RoboDK station: Project.rdk

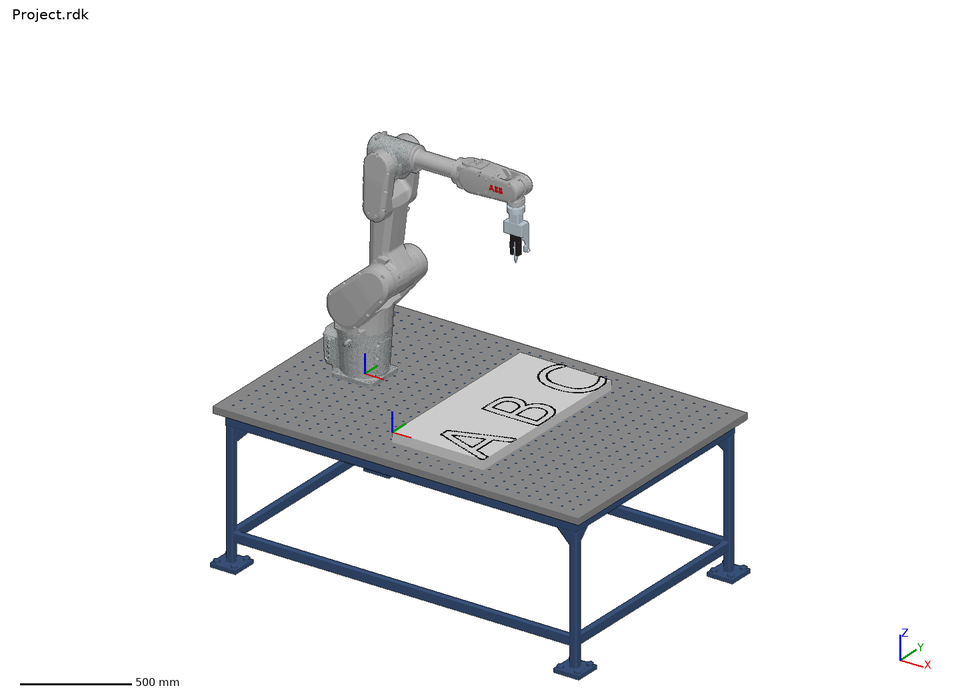
[picture v0: the station drawn from its stored meshes, robots at their saved joint values, targets as dots, program paths as lines]
Station Project (saved by RoboDK 5.5.2). Poses are relative to the parent item; angles as X-Y-Z fixed-axis rotations.
  - object Table at (0, 0, 0) mm, size 2020 x 1340 x 800 mm, geometry from Table-2000x1200x800mm.sld
  - frame Robot_Base at (0, 0, 0) mm
    - robot Robot (model ABB IRB 1300-7/1.4): 6 axes, payload 7 kg, reach 1400 mm, repeatability 0.02 mm, weight 78.5 kg
        modified DH rows (alpha deg, a mm, theta deg, d mm): 0, 0, 0, 544; -90, 150, -90, 0; 0, 575, 0, 0; -90, 40, 0, 675; 90, 0, 0, 0; -90, 0, 180, 90
        joint limits [-180, -95, -210, -230, -130, -400] to [180, 155, 69, 230, 130, 400]; home [0, 0, 0, 0, 0, 0]; saved at [0, 0, 0, 0, 90, 0]
      - tool Pencil, TCP at (0, 0, 283) mm, size 100 x 89.2 x 281.5 mm
    - object pixel at (0, 0, 0) mm, size 10 x 10 x 1 mm
    - frame Board_Frame at (500, -500, 50) mm
      - object Paper_Pixel at (0, 0, 0) mm, size 250 x 250 x 50 mm
      - object Papers at (0, 0, 0) mm, size 505.1 x 1012 x 51 mm
  - Python program main (listed below)

--- Python program main ---
#!/usr/bin/python

# Type help("robodk.robolink") or help("robodk.robomath") for more information
# Press F5 to run the script
# Documentation: https://robodk.com/doc/en/RoboDK-API.html
# Reference:     https://robodk.com/doc/en/PythonAPI/robodk.html
# Note: It is not required to keep a copy of this file, your Python script is saved with your RDK project

# RoboWriter class is a sample class for writing robot.
# For now it assumes that the writing board lies within the robot dextrous workspace

# Import the APIs (RoboDK and Robolink)
from robodk import *
from robolink import *

import sys
import os
import re

SIZE_BOARD = [500, 1000]     # Size of the image. The image will be scaled keeping its aspect ratio
MM_X_PIXEL = 10             # in mm. The path will be cut depending on the pixel size. If this value is changed it is recommended to scale the pixel object

TEXT_SVG='images/test.svg'

class RoboWriter:
    def __init__(self):
        RDK = Robolink()    # Open connection with Robolink library

        # get the robot, frame and tool objects
        self.robot = RDK.Item('', ITEM_TYPE_ROBOT)  # Get the first robot
        self.Board_Frame = RDK.Item('Board_Frame')  # Get the Board_frame
        self.Pencil = RDK.Item('Pencil')            # Get the Pencil

        self.pixel = RDK.Item('pixel')  # get the pixel reference to draw

        image = RDK.Item('Papers')                                   # Get the Paper
        if image.Valid() and image.Type() == ITEM_TYPE_OBJECT:          # If something is already written on the board erase it.
            image.Delete()

        board_pixel = RDK.Item('Paper_Pixel')   # Get the White Board (The display board will be traced using this board)
        # Create Display Board. Difference between White Board and Display board is that
        # White board is a small sized pixel that will be replicated on Display board to
        # show the image

        # Create Display board
        board_pixel.Copy()  # Create a copy of blackboard
        self.board = self.Board_Frame.Paste()   # Create a board with Board Frame as reference frame
        self.board.setVisible(True, False)  # Set the visibility of the board
        self.board.setName('Papers') # Name the board as Display Board

    def write(self, content):
        APPROACH = 100  # approach distance in MM for each path

        home_joints = self.robot.JointsHome().tolist() #[0,0,0,0,90,0] # home joints, in deg
        if abs(home_joints[4]) < 5:
            home_joints[4] = 90.0
        #home_joints[5] = 180

        self.robot.setPoseFrame(self.Board_Frame)
        self.robot.setPoseTool(self.Pencil)
        self.robot.MoveJ(home_joints)   # Move robot to home configuration

        # Get the target orientation depending on the tool orientation at home position
        board_frame_pose = self.Board_Frame.Pose() # Board Frame Pose wrt Robot Base
        robot_flange_pose = self.robot.SolveFK(home_joints) # Robot Flange Pose wrt Robot Base
        TCP_pose = self.Pencil.Pose()   # TCP Pose wrt Flange
        # Use trandformation to get the target orientation wrt Tool
        T2T_Orientation = invH(board_frame_pose)*robot_flange_pose*TCP_pose
        T2T_Orientation[0:3,3] = Mat([0,0,0]) # Set translation to 0

        size_img = content.size_poly()  # returns the size of the current polygon
        self.board.Scale([SIZE_BOARD[0]/250, SIZE_BOARD[1]/250, 1]) # adjust the board size to the image size (scale)

        for path in content:
            # use the pixel reference to set the path color, set pixel width and copy as a reference
            self.pixel.Recolor(path.fill_color)
            data_points_in_current_path = path.nPoints()

            # robot movement: approach to the first target
            initial_target = path.getPoint(0)
            target0 = transl(SIZE_BOARD[0]-initial_target.x, initial_target.y, 0)*T2T_Orientation
            target0_app = target0*transl(0,0,-APPROACH)
            self.robot.MoveL(target0_app)

            for i in range(data_points_in_current_path):
                p_i = path.getPoint(i)
                v_i = path.getVector(i)
                pt_pose = transl(SIZE_BOARD[0]-p_i.x, p_i.y, 0)*rotz(v_i.angle())

                target = transl(SIZE_BOARD[0]-p_i.x, p_i.y, 0)*(T2T_Orientation)

                # Move the robot to the next target
                self.robot.MoveL(target)

                # create a new pixel object with the calculated pixel pose
                self.board.AddGeometry(self.pixel, pt_pose)

            target_app = target*transl(0,0,-APPROACH)
            self.robot.MoveL(target_app)

        self.robot.MoveL(home_joints)

# You can also use the new version of the API:
from svgpy.svg import *
#--------------------------------------------------------------------------------
# Program start
# select the file to draw
# import the SVG file
svgdata = svg_load(TEXT_SVG)

IMAGE_SIZE = Point(SIZE_BOARD[0],SIZE_BOARD[1])   # size of the image in MM
svgdata.calc_polygon_fit(IMAGE_SIZE, MM_X_PIXEL)

writer = RoboWriter()

# draw the image with the robot:
writer.write(svgdata)
